	W =     2.647 deg,	P =   -31.291 deg,	R =   -11.601 deg
   GP2:
	UF : 1, UT : 1,
	J1=   180.000 deg,	J2=  -150.000 deg
};
P[684]{
   GP1:
	UF : 1, UT : 1,		CONFIG : 'N U T, 0, 0, 0',
	X =   799.244  mm,	Y = -1202.971  mm,	Z =  1035.322  mm,
	W =    24.190 deg,	P =   -39.178 deg,	R =    -6.255 deg
   GP2:
	UF : 1, UT : 1,
	J1=   180.000 deg,	J2=  -150.000 deg
};
P[685]{
   GP1:
	UF : 1, UT : 1,		CONFIG : 'N U T, 0, 0, 0',
	X =   954.244  mm,	Y = -1102.971  mm,	Z =   861.322  mm,
	W =    24.190 deg,	P =   -39.178 deg,	R =    -6.255 deg
   GP2:
	UF : 1, UT : 1,
	J1=   180.000 deg,	J2=  -150.000 deg
};
P[686]{
   GP1:
	UF : 1, UT : 1,		CONFIG : 'N U T, 0, 0, 0',
	X =  2596.806  mm,	Y =   482.720  mm,	Z =   -84.201  mm,
	W =   -17.689 deg,	P =    33.470 deg,	R =   110.380 deg
   GP2:
	UF : 1, UT : 1,
	J1=    80.000 deg,	J2=   -90.000 deg
};
P[687]{
   GP1:
	UF : 1, UT : 1,		CONFIG : 'N U T, 0, 0, 0',
	X =  2612.190  mm,	Y =   520.623  mm,	Z =   -86.200  mm,
	W =   -28.177 deg,	P =    11.268 deg,	R =   110.033 deg
   GP2:
	UF : 1, UT : 1,
	J1=    80.000 deg,	J2=   -90.000 deg
};
P[688]{
   GP1:
	UF : 1, UT : 1,		CONFIG : 'N U T, 0, 0, 0',
	X =   955.526  mm,	Y = -1174.727  mm,	Z =   902.888  mm,
	W =    27.863 deg,	P =   -46.318 deg,	R =   -16.260 deg
   GP2:
	UF : 1, UT : 1,
	J1=   180.000 deg,	J2=  -150.000 deg
};
P[689]{
   GP1:
	UF : 1, UT : 1,		CONFIG : 'N U T, 0, 0, 0',
	X =   571.093  mm,	Y = -1097.630  mm,	Z =  1035.072  mm,
	W =    42.871 deg,	P =   -15.240 deg,	R =   -45.029 deg
   GP2:
	UF : 1, UT : 1,
	J1=   180.000 deg,	J2=  -150.000 deg
};
P[690]{
   GP1:
	UF : 1, UT : 1,		CONFIG : 'N U T, 0, 0, 0',
	X =   749.093  mm,	Y =  -654.630  mm,	Z =   835.073  mm,
	W =    44.064 deg,	P =   -10.243 deg,	R =   -50.428 deg
   GP2:
	UF : 1, UT : 1,
	J1=   180.000 deg,	J2=  -150.000 deg
};
P[691]{
   GP1:
	UF : 1, UT : 1,		CONFIG : 'N U T, 0, 0, 0',
	X =  2613.455  mm,	Y =   715.399  mm,	Z =   -86.568  mm,
	W =   -28.922 deg,	P =    12.964 deg,	R =   109.018 deg
   GP2:
	UF : 1, UT : 1,
	J1=    80.000 deg,	J2=   -90.000 deg
};
P[692]{
   GP1:
	UF : 1, UT : 1,		CONFIG : 'N U T, 0, 0, 0',
	X =  2615.403  mm,	Y =   722.950  mm,	Z =   -86.606  mm,
	W =   -28.916 deg,	P =    12.966 deg,	R =    86.670 deg
   GP2:
	UF : 1, UT : 1,
	J1=    80.000 deg,	J2=   -90.000 deg
};
P[693]{
   GP1:
	UF : 1, UT : 1,		CONFIG : 'N U T, 0, 0, 0',
	X =  2616.713  mm,	Y =   727.087  mm,	Z =   -86.606  mm,
	W =   -28.919 deg,	P =    12.966 deg,	R =    81.296 deg
   GP2:
	UF : 1, UT : 1,
	J1=    80.000 deg,	J2=   -90.000 deg
};
P[694]{
   GP1:
	UF : 1, UT : 1,		CONFIG : 'N U T, 0, 0, 0',
	X =   962.545  mm,	Y = -1093.036  mm,	Z =   867.966  mm,
	W =    44.863 deg,	P =     3.974 deg,	R =   -63.984 deg
   GP2:
	UF : 1, UT : 1,
	J1=   180.000 deg,	J2=  -150.000 deg
};
P[695]{
   GP1:
	UF : 1, UT : 1,		CONFIG : 'N U T, 0, 0, 0',
	X =   592.698  mm,	Y =  -634.536  mm,	Z =   863.966  mm,
	W =    36.388 deg,	P =   -28.554 deg,	R =   -27.033 deg
   GP2:
	UF : 1, UT : 1,
	J1=   180.000 deg,	J2=  -150.000 deg
};
P[696]{
   GP1:
	UF : 1, UT : 1,		CONFIG : 'N U T, 0, 0, 0',
	X =  2624.650  mm,	Y =   752.415  mm,	Z =   -87.415  mm,
	W =   -29.838 deg,	P =     9.278 deg,	R =    96.979 deg
   GP2:
	UF : 1, UT : 1,
	J1=    80.000 deg,	J2=   -90.000 deg
};
P[697]{
   GP1:
	UF : 1, UT : 1,		CONFIG : 'N U T, 0, 0, 0',
	X =  2621.804  mm,	Y =   771.484  mm,	Z =   -88.918  mm,
	W =   -33.766 deg,	P =      .741 deg,	R =   119.819 deg
   GP2:
	UF : 1, UT : 1,
	J1=    80.000 deg,	J2=   -90.000 deg
};
P[698]{
   GP1:
	UF : 1, UT : 1,		CONFIG : 'N U T, 0, 0, 0',
	X =   545.804  mm,	Y =  -597.246  mm,	Z =   979.702  mm,
	W =    15.937 deg,	P =   -42.493 deg,	R =     6.853 deg
   GP2:
	UF : 1, UT : 1,
	J1=   180.000 deg,	J2=  -150.000 deg
};
P[699]{
   GP1:
	UF : 1, UT : 1,		CONFIG : 'N U T, 0, 0, 0',
	X =   366.532  mm,	Y =  -833.172  mm,	Z =  1480.397  mm,
	W =    13.558 deg,	P =     8.679 deg,	R =   -55.514 deg
   GP2:
	UF : 1, UT : 1,
	J1=   180.000 deg,	J2=  -150.000 deg
};
P[700]{
   GP1:
	UF : 1, UT : 1,		CONFIG : 'N U T, 0, 0, 0',
	X =  1532.562  mm,	Y = -1156.369  mm,	Z =  1523.814  mm,
	W =   -53.323 deg,	P =    -7.912 deg,	R =   -20.862 deg
   GP2:
	UF : 0, UT : 1,
	J1=   180.000 deg,	J2=   -90.000 deg
};
P[701]{
   GP1:
	UF : 1, UT : 1,		CONFIG : 'N U T, 0, 0, 0',
	X =  1863.519  mm,	Y = -1304.565  mm,	Z =  1265.460  mm,
	W =   -45.547 deg,	P =    -6.107 deg,	R =    -5.943 deg
   GP2:
	UF : 0, UT : 1,
	J1=   180.000 deg,	J2=   -90.000 deg
};
P[702]{
   GP1:
	UF : 1, UT : 1,		CONFIG : 'N U T, 0, 0, 0',
	X =  1929.519  mm,	Y = -1405.565  mm,	Z =  1058.460  mm,
	W =   -42.701 deg,	P =    18.644 deg,	R =    19.122 deg
   GP2:
	UF : 0, UT : 1,
	J1=   180.000 deg,	J2=   -90.000 deg
};
P[703]{
   GP1:
	UF : 1, UT : 1,		CONFIG : 'N U T, 0, 0, 0',
	X =  2567.091  mm,	Y =   800.104  mm,	Z =   -75.608  mm,
	W =    -3.304 deg,	P =   -34.460 deg,	R =   105.018 deg
   GP2:
	UF : 1, UT : 1,
	J1=    80.000 deg,	J2=   -90.000 deg
};
P[704]{
   GP1:
	UF : 1, UT : 1,		CONFIG : 'N U T, 0, 0, 0',
	X =  2590.479  mm,	Y =   800.309  mm,	Z =   -79.339  mm,
	W =    -3.314 deg,	P =   -34.462 deg,	R =   105.031 deg
   GP2:
	UF : 1, UT : 1,
	J1=    80.000 deg,	J2=   -90.000 deg
};
P[705]{
   GP1:
	UF : 1, UT : 1,		CONFIG : 'N U T, 0, 0, 0',
	X =  2605.620  mm,	Y =   794.752  mm,	Z =   -80.490  mm,
	W =     3.036 deg,	P =   -34.484 deg,	R =    65.941 deg
   GP2:
	UF : 1, UT : 1,
	J1=    80.000 deg,	J2=   -90.000 deg
};
P[706]{
   GP1:
	UF : 1, UT : 1,		CONFIG : 'N U T, 0, 0, 0',
	X =  2628.806  mm,	Y =   769.334  mm,	Z =   -84.912  mm,
	W =   -11.646 deg,	P =   -32.810 deg,	R =    38.711 deg
   GP2:
	UF : 1, UT : 1,
	J1=    80.000 deg,	J2=   -90.000 deg
};
P[708]{
   GP1:
	UF : 1, UT : 1,		CONFIG : 'N U T, 0, 0, 0',
	X =  2039.010  mm,	Y = -1381.508  mm,	Z =  1071.568  mm,
	W =   -44.862 deg,	P =     3.961 deg,	R =   -20.537 deg
   GP2:
	UF : 0, UT : 1,
	J1=   180.000 deg,	J2=   -90.000 deg
};
P[710]{
   GP1:
	UF : 1, UT : 1,		CONFIG : 'N U T, 0, 0, 0',
	X =  1822.564  mm,	Y = -1057.861  mm,	Z =  1463.123  mm,
	W =   -36.308 deg,	P =    -6.286 deg,	R =   -23.397 deg
   GP2:
	UF : 1, UT : 1,
	J1=   180.000 deg,	J2=   -90.000 deg
};
P[711]{
   GP1:
	UF : 1, UT : 1,		CONFIG : 'N U T, 0, 0, 0',
	X =  1392.804  mm,	Y =   640.782  mm,	Z =  1670.105  mm,
	W =    37.735 deg,	P =   -20.539 deg,	R =     -.894 deg
   GP2:
	UF : 0, UT : 1,
	J1=   180.000 deg,	J2=    90.000 deg
};
P[712]{
   GP1:
	UF : 1, UT : 1,		CONFIG : 'N U T, 0, 0, 0',
	X =  1849.519  mm,	Y =  1220.906  mm,	Z =  1351.461  mm,
	W =    44.958 deg,	P =    -2.212 deg,	R =     2.229 deg
   GP2:
	UF : 0, UT : 1,
	J1=   180.000 deg,	J2=    90.000 deg
};
P[713]{
   GP1:
	UF : 1, UT : 1,		CONFIG : 'N U T, 0, 0, 0',
	X =  1880.451  mm,	Y =  1275.016  mm,	Z =  1238.303  mm,
	W =    44.592 deg,	P =     6.805 deg,	R =    -6.838 deg
   GP2:
	UF : 1, UT : 1,
	J1=   180.000 deg,	J2=    90.000 deg
};
P[714]{
   GP1:
	UF : 1, UT : 1,		CONFIG : 'N U T, 0, 0, 0',
	X =  1926.400  mm,	Y =  1355.399  mm,	Z =  1070.204  mm,
	W =    41.277 deg,	P =    19.800 deg,	R =   -21.086 deg
   GP2:
	UF : 0, UT : 1,
	J1=   180.000 deg,	J2=    90.000 deg
};
P[716]{
   GP1:
	UF : 1, UT : 1,		CONFIG : 'N U T, 0, 0, 0',
	X =  1054.944  mm,	Y = -1059.833  mm,	Z =   786.244  mm,
	W =    24.545 deg,	P =   -38.987 deg,	R =    -6.159 deg
   GP2:
	UF : 1, UT : 1,
	J1=   180.000 deg,	J2=  -150.000 deg
};
P[717]{
   GP1:
	UF : 1, UT : 1,		CONFIG : 'N U T, 0, 0, 0',
	X =  1096.676  mm,	Y = -1131.783  mm,	Z =   786.792  mm,
	W =    24.536 deg,	P =   -38.987 deg,	R =    -6.145 deg
   GP2:
	UF : 1, UT : 1,
	J1=   180.000 deg,	J2=  -150.000 deg
};
P[718]{
   GP1:
	UF : 1, UT : 1,		CONFIG : 'N U T, 0, 0, 0',
	X =   775.910  mm,	Y =  -578.708  mm,	Z =   787.478  mm,
	W =    38.781 deg,	P =   -22.219 deg,	R =   -34.485 deg
   GP2:
	UF : 1, UT : 1,
	J1=   180.000 deg,	J2=  -150.000 deg
};
P[719]{
   GP1:
	UF : 1, UT : 1,		CONFIG : 'N U T, 0, 0, 0',
	X =   809.929  mm,	Y =  -635.718  mm,	Z =   787.471  mm,
	W =    42.821 deg,	P =    -9.985 deg,	R =   -50.263 deg
   GP2:
	UF : 1, UT : 1,
	J1=   180.000 deg,	J2=  -150.000 deg
};
P[720]{
   GP1:
	UF : 1, UT : 1,		CONFIG : 'N U T, 0, 0, 0',
	X =  1993.007  mm,	Y =  1431.170  mm,	Z =  1068.677  mm,
	W =    44.305 deg,	P =     8.850 deg,	R =     3.803 deg
   GP2:
	UF : 1, UT : 1,
	J1=   180.000 deg,	J2=    90.000 deg
};
P[721]{
   GP1:
	UF : 1, UT : 1,		CONFIG : 'N U T, 0, 0, 0',
	X =  1840.948  mm,	Y =  1174.835  mm,	Z =  1330.032  mm,
	W =    44.958 deg,	P =    -2.212 deg,	R =     2.229 deg
   GP2:
	UF : 0, UT : 1,
	J1=   180.000 deg,	J2=    90.000 deg
};
P[723]{
   GP1:
	UF : 1, UT : 1,		CONFIG : 'N U T, 0, 0, 0',
	X =   914.639  mm,	Y =  -816.989  mm,	Z =   784.680  mm,
	W =    43.515 deg,	P =    -5.259 deg,	R =   -59.147 deg
   GP2:
	UF : 1, UT : 1,
	J1=   180.000 deg,	J2=  -150.000 deg
};
P[724]{
   GP1:
	UF : 1, UT : 1,		CONFIG : 'N U T, 0, 0, 0',
	X =  1031.765  mm,	Y = -1020.352  mm,	Z =   782.958  mm,
	W =    42.900 deg,	P =    -9.647 deg,	R =   -54.444 deg
   GP2:
	UF : 1, UT : 1,
	J1=   180.000 deg,	J2=  -150.000 deg
};
P[725]{
   GP1:
	UF : 1, UT : 1,		CONFIG : 'N U T, 0, 0, 0',
	X =   756.230  mm,	Y =  -541.089  mm,	Z =   785.795  mm,
	W =    29.846 deg,	P =   -35.386 deg,	R =   -14.750 deg
   GP2:
	UF : 1, UT : 1,
	J1=   180.000 deg,	J2=  -150.000 deg
};
P[726]{
   GP1:
	UF : 1, UT : 1,		CONFIG : 'N U T, 0, 0, 0',
	X =   729.622  mm,	Y =  -504.659  mm,	Z =   786.044  mm,
	W =     5.274 deg,	P =   -44.804 deg,	R =    22.436 deg
   GP2:
	UF : 1, UT : 1,
	J1=   179.999 deg,	J2=  -150.000 deg
};
P[727]{
   GP1:
	UF : 1, UT : 1,		CONFIG : 'N U T, 0, 0, 0',
	X =  1896.353  mm,	Y = -1475.130  mm,	Z =  1030.048  mm,
	W =   -39.886 deg,	P =    23.867 deg,	R =    23.914 deg
   GP2:
	UF : 1, UT : 1,
	J1=   180.000 deg,	J2=   -90.000 deg
};
P[728]{
   GP1:
	UF : 1, UT : 1,		CONFIG : 'N U T, 0, 0, 0',
	X =  1926.846  mm,	Y = -1474.183  mm,	Z =  1030.788  mm,
	W =   -43.541 deg,	P =    14.556 deg,	R =    14.831 deg
   GP2:
	UF : 1, UT : 1,
	J1=   180.000 deg,	J2=   -90.000 deg
};
P[729]{
   GP1:
	UF : 1, UT : 1,		CONFIG : 'N U T, 0, 0, 0',
	X =  1957.542  mm,	Y = -1475.449  mm,	Z =  1029.331  mm,
	W =   -43.543 deg,	P =    14.555 deg,	R =    14.822 deg
   GP2:
	UF : 1, UT : 1,
	J1=   180.000 deg,	J2=   -90.000 deg
};
P[730]{
   GP1:
	UF : 1, UT : 1,		CONFIG : 'N U T, 0, 0, 0',
	X =  1986.256  mm,	Y = -1488.593  mm,	Z =  1028.687  mm,
	W =   -43.543 deg,	P =    14.555 deg,	R =   -14.019 deg
   GP2:
	UF : 1, UT : 1,
	J1=   180.000 deg,	J2=   -90.000 deg
};
P[731]{
   GP1:
	UF : 1, UT : 1,		CONFIG : 'N U T, 0, 0, 0',
	X =  1996.570  mm,	Y = -1499.152  mm,	Z =  1027.769  mm,
	W =   -44.808 deg,	P =     8.519 deg,	R =   -27.703 deg
   GP2:
	UF : 1, UT : 1,
	J1=   180.000 deg,	J2=   -90.000 deg
};
P[732]{
   GP1:
	UF : 1, UT : 1,		CONFIG : 'F U T, 0, 0, 0',
	X =   804.374  mm,	Y =   981.069  mm,	Z =  1117.927  mm,
	W =    50.730 deg,	P =      .639 deg,	R =   -51.736 deg
   GP2:
	UF : 1, UT : 1,
	J1=   180.000 deg,	J2=   150.000 deg
};
P[733]{
   GP1:
	UF : 1, UT : 1,		CONFIG : 'F U T, 0, 0, 0',
	X =  1064.016  mm,	Y =   999.283  mm,	Z =  1072.926  mm,
	W =    50.730 deg,	P =      .639 deg,	R =   -51.736 deg
   GP2:
	UF : 1, UT : 1,
	J1=   180.000 deg,	J2=   150.000 deg
};
P[734]{
   GP1:
	UF : 1, UT : 1,		CONFIG : 'N U T, 0, 0, 0',
	X =  1905.120  mm,	Y =  1477.933  mm,	Z =  1024.903  mm,
	W =    41.277 deg,	P =    19.801 deg,	R =   -17.230 deg
   GP2:
	UF : 1, UT : 1,
	J1=   180.000 deg,	J2=    90.000 deg
};
P[735]{
   GP1:
	UF : 1, UT : 1,		CONFIG : 'N U T, 0, 0, 0',
	X =  1928.835  mm,	Y =  1475.574  mm,	Z =  1026.258  mm,
	W =    41.277 deg,	P =    19.801 deg,	R =   -17.230 deg
   GP2:
	UF : 1, UT : 1,
	J1=   180.000 deg,	J2=    90.000 deg
};
P[736]{
   GP1:
	UF : 1, UT : 1,		CONFIG : 'N U T, 0, 0, 0',
	X =  1969.406  mm,	Y =  1474.718  mm,	Z =  1027.759  mm,
	W =    41.277 deg,	P =    19.801 deg,	R =   -17.230 deg
   GP2:
	UF : 1, UT : 1,
	J1=   180.000 deg,	J2=    90.000 deg
};
P[737]{
   GP1:
	UF : 1, UT : 1,		CONFIG : 'N U T, 0, 0, 0',
	X =  1984.906  mm,	Y =  1480.576  mm,	Z =  1025.115  mm,
	W =    41.276 deg,	P =    19.801 deg,	R =     6.735 deg
   GP2:
	UF : 1, UT : 1,
	J1=   180.000 deg,	J2=    90.000 deg
};
P[738]{
   GP1:
	UF : 1, UT : 1,		CONFIG : 'F U T, 0, 0, 0',
	X =  1102.958  mm,	Y =   975.094  mm,	Z =  1056.986  mm,
	W =    50.535 deg,	P =   -23.426 deg,	R =   -25.981 deg
   GP2:
	UF : 1, UT : 1,
	J1=   180.000 deg,	J2=   150.000 deg
};
P[739]{
   GP1:
	UF : 1, UT : 1,		CONFIG : 'F U T, 0, 0, 0',
	X =   851.887  mm,	Y =   977.237  mm,	Z =  1067.701  mm,
	W =    50.535 deg,	P =   -23.426 deg,	R =   -25.981 deg
   GP2:
	UF : 1, UT : 1,
	J1=   180.000 deg,	J2=   150.000 deg
};
P[740]{
   GP1:
	UF : 1, UT : 1,		CONFIG : 'F U T, 0, 0, 0',
	X =   626.208  mm,	Y =  1096.450  mm,	Z =  1381.774  mm,
	W =    61.728 deg,	P =   -31.893 deg,	R =   -10.883 deg
   GP2:
	UF : 1, UT : 1,
	J1=   180.000 deg,	J2=   150.000 deg
};
P[741]{
   GP1:
	UF : 1, UT : 1,		CONFIG : 'N U T, 0, 0, 0',
	X =  1998.833  mm,	Y =  1491.079  mm,	Z =  1024.830  mm,
	W =    43.864 deg,	P =    11.266 deg,	R =    16.926 deg
   GP2:
	UF : 1, UT : 1,
	J1=   180.000 deg,	J2=    90.000 deg
};
P[742]{
   GP1:
	UF : 1, UT : 1,		CONFIG : 'N U T, 0, 0, 0',
	X =  1640.567  mm,	Y = -1414.013  mm,	Z =  1035.421  mm,
	W =   -42.856 deg,	P =   -15.294 deg,	R =    39.130 deg
   GP2:
	UF : 1, UT : 1,
	J1=   180.000 deg,	J2=  -125.000 deg
};
P[743]{
   GP1:
	UF : 1, UT : 1,		CONFIG : 'N U T, 0, 0, 0',
	X =  1646.214  mm,	Y = -1407.571  mm,	Z =  1034.707  mm,
	W =   -42.573 deg,	P =   -16.796 deg,	R =    40.474 deg
   GP2:
	UF : 1, UT : 1,
	J1=   180.000 deg,	J2=  -125.000 deg
};
P[744]{
   GP1:
	UF : 1, UT : 1,		CONFIG : 'N U T, 0, 0, 0',
	X =  1661.285  mm,	Y = -1395.356  mm,	Z =  1034.707  mm,
	W =   -42.573 deg,	P =   -16.796 deg,	R =    43.536 deg
   GP2:
	UF : 1, UT : 1,
	J1=   180.000 deg,	J2=  -125.000 deg
};
P[745]{
   GP1:
	UF : 1, UT : 1,		CONFIG : 'N U T, 0, 0, 0',
	X =  1683.971  mm,	Y = -1387.000  mm,	Z =  1035.270  mm,
	W =   -44.235 deg,	P =   -18.485 deg,	R =    48.309 deg
   GP2:
	UF : 1, UT : 1,
	J1=   180.000 deg,	J2=  -125.000 deg
};
P[746]{
   GP1:
	UF : 1, UT : 1,		CONFIG : 'F U T, 0, 0, 0',
	X =  1108.465  mm,	Y =  1009.734  mm,	Z =  1037.331  mm,
	W =    45.728 deg,	P =    -4.747 deg,	R =   -51.700 deg
   GP2:
	UF : 1, UT : 1,
	J1=   180.000 deg,	J2=   150.000 deg
};
P[747]{
   GP1:
	UF : 1, UT : 1,		CONFIG : 'F U T, 0, 0, 0',
	X =  1119.770  mm,	Y =  1005.438  mm,	Z =  1036.133  mm,
	W =    42.645 deg,	P =    -7.518 deg,	R =   -34.906 deg
   GP2:
	UF : 1, UT : 1,
	J1=   180.000 deg,	J2=   150.000 deg
};
P[748]{
   GP1:
	UF : 1, UT : 1,		CONFIG : 'F U T, 0, 0, 0',
	X =  1137.596  mm,	Y =  1002.274  mm,	Z =  1035.866  mm,
	W =    42.486 deg,	P =   -15.624 deg,	R =   -17.645 deg
   GP2:
	UF : 1, UT : 1,
	J1=   180.000 deg,	J2=   150.000 deg
};
P[749]{
   GP1:
	UF : 1, UT : 1,		CONFIG : 'F U T, 0, 0, 0',
	X =  1149.397  mm,	Y =  1000.482  mm,	Z =  1037.765  mm,
	W =    42.477 deg,	P =   -15.634 deg,	R =   -23.232 deg
   GP2:
	UF : 1, UT : 1,
	J1=   180.000 deg,	J2=   150.000 deg
};
P[768]{
   GP1:
	UF : 1, UT : 1,		CONFIG : 'N U T, 0, 0, 0',
	X =  1082.860  mm,	Y =     -.638  mm,	Z =   529.898  mm,
	W =    48.292 deg,	P =    28.213 deg,	R =    20.411 deg
   GP2:
	UF : 1, UT : 1,
	J1=    80.000 deg,	J2=    90.000 deg
};
P[775]{
   GP1:
	UF : 1, UT : 1,		CONFIG : 'N U T, 0, 0, 0',
	X =  2345.678  mm,	Y =   -89.733  mm,	Z =   -12.555  mm,
	W =    43.244 deg,	P =    13.889 deg,	R =   -17.216 deg
   GP2:
	UF : 1, UT : 1,
	J1=    90.000 deg,	J2=    90.000 deg
};
P[776]{
   GP1:
	UF : 1, UT : 1,		CONFIG : 'N U T, 0, 0, 0',
	X =  2390.535  mm,	Y =   -88.876  mm,	Z =   -12.554  mm,
	W =    43.244 deg,	P =    13.889 deg,	R =   -17.216 deg
   GP2:
	UF : 1, UT : 1,
	J1=    90.000 deg,	J2=    90.000 deg
};
P[777]{
   GP1:
	UF : 1, UT : 1,		CONFIG : 'N U T, 0, 0, 0',
	X =  2413.115  mm,	Y =   -88.080  mm,	Z =   -11.207  mm,
	W =    43.008 deg,	P =    13.906 deg,	R =   -45.606 deg
   GP2:
	UF : 1, UT : 1,
	J1=    89.995 deg,	J2=    90.000 deg
};
P[793]{
   GP1:
	UF : 1, UT : 1,		CONFIG : 'F U T, 0, 0, 0',
	X =   419.331  mm,	Y =  1026.789  mm,	Z =  1609.020  mm,
	W =    71.318 deg,	P =     7.769 deg,	R =   -20.454 deg
   GP2:
	UF : 1, UT : 1,
	J1=   180.000 deg,	J2=   150.000 deg
};
/END
